Fanuc KAREL source: ka00185.KL

-- PROVISIONAL review KL for V1013-1; original PC SHA256 4198479cfcb88fec3e39e292a4df897bb08ce01634c3d37d88b3fc821ff398df
-- Incomplete behavior may be omitted. Consult companion uncertainty JSON. Do not deploy.
PROGRAM KA00185
%NOLOCKGROUP
-- UNRESOLVED_DECL SRC type=002018
-- UNRESOLVED_DECL DST type=002018
BEGIN
  -- UNRESOLVED_PC offsets 5-19; opcodes 22,22,1E
  -- UNRESOLVED_PC offsets 24-28; opcodes 7F
END KA00185
